FUNCTION_BLOCK "Swan_AMI_pH-Redox"   // FB69, SCL
{ S7_Optimized_Access := 'TRUE' }
VERSION : 0.1
   VAR_INPUT
      mb_addr : USInt;
   END_VAR
   VAR_IN_OUT
      mb_query : "mb_query";
   END_VAR
   VAR
      sb : "mb_station_block_udt";
      data : Struct
         pH_Redox : Real;   // pH/mV
         temperature : Real;   // °C
         Flow : Real;   // l/h
         raw_signal : Real;   // mV
         Pt_1000_temp : Real;   // ohm
         raw_flow : Real;   // Hz
         sensor_check : Real;   // Mohm
         case_temperature : Real;   // °C
         signal_output_1 : Real;   // mA
         signal_output_2 : Real;   // mA
         instrument_display_status : DWord;
      END_STRUCT;
      alarm : Struct
         x00_alarm_high : Bool;
         x01_alarm_low : Bool;
         x02 : Bool;
         x03 : Bool;
         x04 : Bool;
         x05 : Bool;
         x06_sample_temp_high : Bool;
         x07_sample_temp_low : Bool;
         x08_sample_flow_high : Bool;
         x09_sample_flow_low : Bool;
         x10_temp_shorted : Bool;
         x11_temp_disconnected : Bool;
         x12_case_temp_high : Bool;
         x13_case_temp_low : Bool;
         x14 : Bool;
         x15 : Bool;
         x16_control_timeout : Bool;
         x17 : Bool;
         x18 : Bool;
         x19 : Bool;
         x20 : Bool;
         x21 : Bool;
         x22 : Bool;
         x23_input_active : Bool;
         x24_IC_MK41T56 : Bool;
         x25_IC_LM75 : Bool;
         x26_IC_PCF8574 : Bool;
         x27_Signal_output_open : Bool;
         x28_EEprom_Motherboard : Bool;
         x29_EEprom_Front_end : Bool;
         x30_Calibration_Recout : Bool;
         x31_Wrong_Front_end : Bool;
      END_STRUCT;
      write : Struct
         x0_relay_contacts_1 : Bool;
         x1_relay_contacts_2 : Bool;
         x2_hold : Bool;
         x3_Remote_off : Bool;
         x4 : Bool;
         x5 : Bool;
         x6 : Bool;
         x7 : Bool;
      END_STRUCT;
   END_VAR
BEGIN
   // Swan - AMI pH-Redox
   // Swan analytical instruments
   // 
   // http://www.swan.ch/GetAttachment.axd?attaName=e82f8e94-ab32-4930-8c9d-a56dc0847f61
   // Page 73

   "mb_station_block_header"(sb := #sb, mb_query := #mb_query);
   #mb_query.mb_addr := #mb_addr;
   #mb_query.data_addr := 0;

   #mb_query(mode := #mb_query.c.read.input_reg,
             data_ptr := #data);

   #mb_query(mode := #mb_query.c.read.discrete_input,
             data_ptr := #alarm);

   (*#mb_query(mode := #mb_query.c.write.discrete_output,
             data_len := 4,
             data_ptr := #write);*)

   "mb_station_block_footer"(sb := #sb, mb_query := #mb_query);
END_FUNCTION_BLOCK

// folder: Library/Modbus/Station blocks/_Extend blocks

FUNCTION_BLOCK "searchDevice"   // FB41, SCL
{ S7_Optimized_Access := 'TRUE' }
VERSION : 0.1
   VAR_OUTPUT
      Done : Bool;
      No_finding : Bool;
   END_VAR
   VAR_IN_OUT
      start_search : Bool;
      mb_addr : UInt;
      mb_query : "mb_query";
   END_VAR
   VAR
      reset_at_start : Bool;
      data_addr : UDInt;
      _ : Bool;
      rtirg_start : R_TRIG;
      resualt_data : Word;
   END_VAR
BEGIN
   #rtirg_start(CLK := #start_search);
   IF #rtirg_start.Q AND #reset_at_start THEN
       #mb_addr := 1;
   END_IF;

   IF #start_search THEN
       #Done := false;
       #No_finding := false;
       #mb_query(mb_addr := #mb_addr,
                 mode := #mb_query.c.read.holding_reg,
                 data_addr := #data_addr,
                 data_ptr := #resualt_data);
       IF #mb_query.Done
           OR #mb_query.Error AND NOT #mb_query.stat.error_comm
       THEN
           #Done := true;
           #start_search := false;
       ELSIF #mb_query.Error THEN
           IF #mb_addr < 247 THEN
               #mb_addr += 1;
           ELSE
               #No_finding := true;
               #start_search := false;
           END_IF;
       END_IF;
   END_IF;
END_FUNCTION_BLOCK

// folder: Library/Modbus/Station blocks/zz Internal special

FUNCTION_BLOCK "temeratur_transmitter"   // FB2, SCL
{ S7_Optimized_Access := 'TRUE' }
VERSION : 0.1
   VAR_OUTPUT
      Temperatur : Real;
   END_VAR
   VAR_IN_OUT
      mb_query : "mb_query";
   END_VAR
   VAR
      sb : "mb_station_block_udt";
   END_VAR
   VAR_TEMP
      tmp : Int;
   END_VAR
BEGIN
   // Temperatur transmitter.

   "mb_station_block_header"(sb := #sb, mb_query := #mb_query);

   #mb_query(mb_addr := 1,
             mode := #mb_query.c.read.holding_reg,
             data_addr := 0,
             data_ptr := #tmp);

   IF #mb_query.Done THEN
       #Temperatur := REAL_TO_INT(#tmp) / 10;
   END_IF;

   "mb_station_block_footer"(sb := #sb, mb_query := #mb_query);
END_FUNCTION_BLOCK